// TIA Portal V18 export
FUNCTION "Pump Management" : Void   // FC44, LAD
{ S7_Optimized_Access := 'TRUE' }
VERSION : 0.1
// stored: AutoNumber false, IsIECCheckEnabled false, SetENOAutomatically false, UDAEnableTagReadback false
   VAR_TEMP
      mbit1 : Bool;
   END_VAR
BEGIN

REGION Network 1
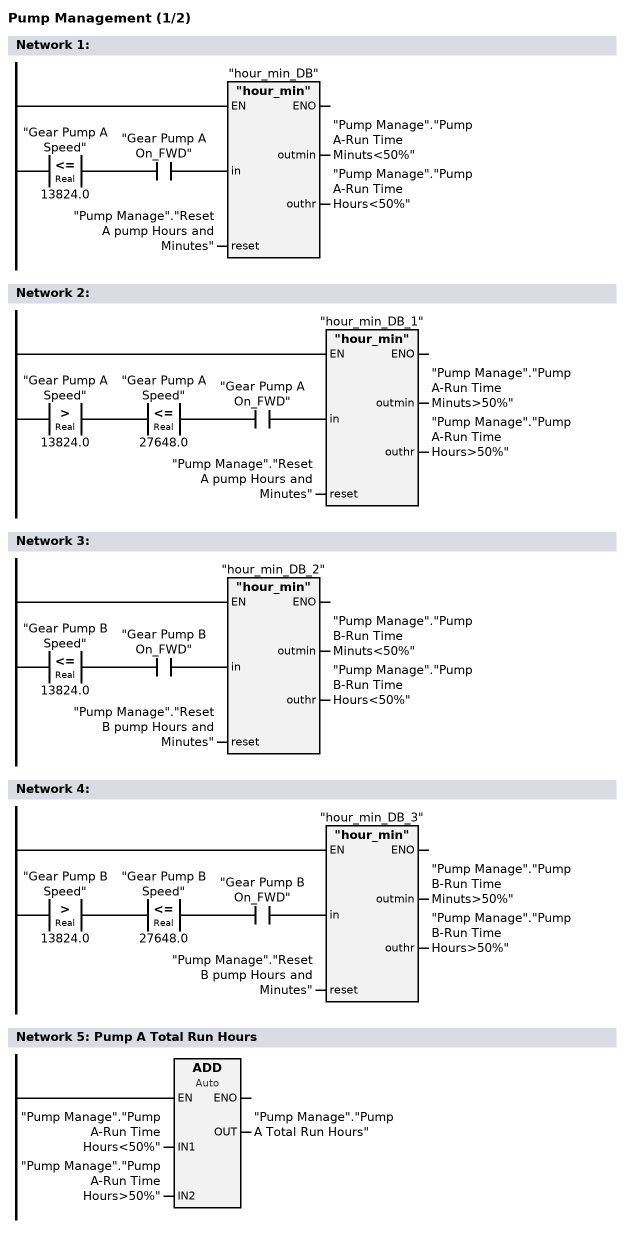
   RUNG wire#powerrail
      "hour_min_DB"(in := wire#w1, reset := "Pump Manage"."Reset A pump Hours and Minutes", outmin => "Pump Manage"."Pump A-Run Time Minuts<50%", outhr => "Pump Manage"."Pump A-Run Time Hours<50%")
   END_RUNG
   RUNG wire#powerrail
      { S7_Templates := "SrcType := Real" } LE_Contact(in1 := "Gear Pump A Speed", in2 := 13824.0)
      Contact( "Gear Pump A On_FWD" )
   END_RUNG wire#w1
   // the same network as SCL:
   "hour_min_DB"(in := ("Gear Pump A Speed" <= 13824.0) AND "Gear Pump A On_FWD",   // "hour_min"
                 reset := "Pump Manage"."Reset A pump Hours and Minutes",
                 outmin => "Pump Manage"."Pump A-Run Time Minuts<50%",
                 outhr => "Pump Manage"."Pump A-Run Time Hours<50%");
END_REGION

REGION Network 2
   RUNG wire#powerrail
      "hour_min_DB_1"(in := wire#w1, reset := "Pump Manage"."Reset A pump Hours and Minutes", outmin => "Pump Manage"."Pump A-Run Time Minuts>50%", outhr => "Pump Manage"."Pump A-Run Time Hours>50%")
   END_RUNG
   RUNG wire#powerrail
      { S7_Templates := "SrcType := Real" } GT_Contact(in1 := "Gear Pump A Speed", in2 := 13824.0)
      { S7_Templates := "SrcType := Real" } LE_Contact(in1 := "Gear Pump A Speed", in2 := 27648.0)
      Contact( "Gear Pump A On_FWD" )
   END_RUNG wire#w1
   // the same network as SCL:
   "hour_min_DB_1"(in := ("Gear Pump A Speed" > 13824.0) AND ("Gear Pump A Speed" <= 27648.0) AND "Gear Pump A On_FWD",   // "hour_min"
                   reset := "Pump Manage"."Reset A pump Hours and Minutes",
                   outmin => "Pump Manage"."Pump A-Run Time Minuts>50%",
                   outhr => "Pump Manage"."Pump A-Run Time Hours>50%");
END_REGION

REGION Network 3
   RUNG wire#powerrail
      "hour_min_DB_2"(in := wire#w1, reset := "Pump Manage"."Reset B pump Hours and Minutes", outmin => "Pump Manage"."Pump B-Run Time Minuts<50%", outhr => "Pump Manage"."Pump B-Run Time Hours<50%")
   END_RUNG
   RUNG wire#powerrail
      { S7_Templates := "SrcType := Real" } LE_Contact(in1 := "Gear Pump B Speed", in2 := 13824.0)
      Contact( "Gear Pump B On_FWD" )
   END_RUNG wire#w1
   // the same network as SCL:
   "hour_min_DB_2"(in := ("Gear Pump B Speed" <= 13824.0) AND "Gear Pump B On_FWD",   // "hour_min"
                   reset := "Pump Manage"."Reset B pump Hours and Minutes",
                   outmin => "Pump Manage"."Pump B-Run Time Minuts<50%",
                   outhr => "Pump Manage"."Pump B-Run Time Hours<50%");
END_REGION

REGION Network 4
   RUNG wire#powerrail
      "hour_min_DB_3"(in := wire#w1, reset := "Pump Manage"."Reset B pump Hours and Minutes", outmin => "Pump Manage"."Pump B-Run Time Minuts>50%", outhr => "Pump Manage"."Pump B-Run Time Hours>50%")
   END_RUNG
   RUNG wire#powerrail
      { S7_Templates := "SrcType := Real" } GT_Contact(in1 := "Gear Pump B Speed", in2 := 13824.0)
      { S7_Templates := "SrcType := Real" } LE_Contact(in1 := "Gear Pump B Speed", in2 := 27648.0)
      Contact( "Gear Pump B On_FWD" )
   END_RUNG wire#w1
   // the same network as SCL:
   "hour_min_DB_3"(in := ("Gear Pump B Speed" > 13824.0) AND ("Gear Pump B Speed" <= 27648.0) AND "Gear Pump B On_FWD",   // "hour_min"
                   reset := "Pump Manage"."Reset B pump Hours and Minutes",
                   outmin => "Pump Manage"."Pump B-Run Time Minuts>50%",
                   outhr => "Pump Manage"."Pump B-Run Time Hours>50%");
END_REGION

REGION Network 5: Pump A Total Run Hours
   RUNG wire#powerrail
      Add(in1 := "Pump Manage"."Pump A-Run Time Hours<50%", in2 := "Pump Manage"."Pump A-Run Time Hours>50%", out => "Pump Manage"."Pump A Total Run Hours")
   END_RUNG
   // the same network as SCL:
   "Pump Manage"."Pump A Total Run Hours" := "Pump Manage"."Pump A-Run Time Hours<50%" + "Pump Manage"."Pump A-Run Time Hours>50%";
END_REGION

REGION Network 6: Pump A Total Run Minutes
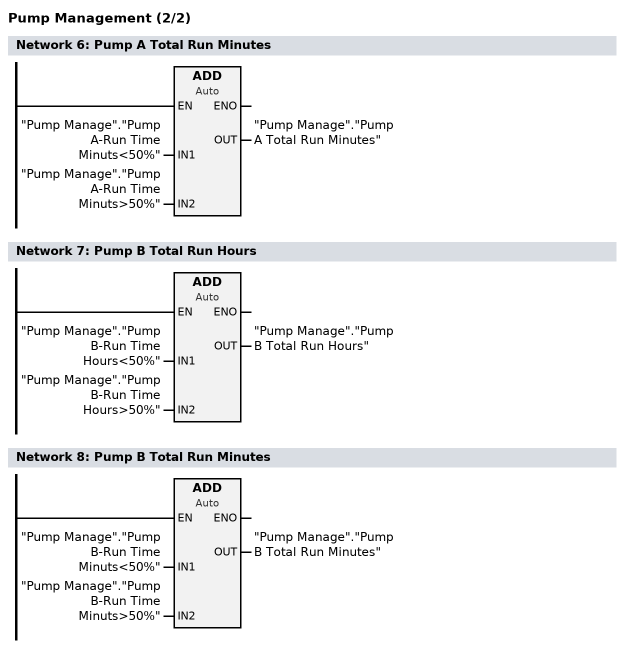
   RUNG wire#powerrail
      Add(in1 := "Pump Manage"."Pump A-Run Time Minuts<50%", in2 := "Pump Manage"."Pump A-Run Time Minuts>50%", out => "Pump Manage"."Pump A Total Run Minutes")
   END_RUNG
   // the same network as SCL:
   "Pump Manage"."Pump A Total Run Minutes" := "Pump Manage"."Pump A-Run Time Minuts<50%" + "Pump Manage"."Pump A-Run Time Minuts>50%";
END_REGION

REGION Network 7: Pump B Total Run Hours
   RUNG wire#powerrail
      Add(in1 := "Pump Manage"."Pump B-Run Time Hours<50%", in2 := "Pump Manage"."Pump B-Run Time Hours>50%", out => "Pump Manage"."Pump B Total Run Hours")
   END_RUNG
   // the same network as SCL:
   "Pump Manage"."Pump B Total Run Hours" := "Pump Manage"."Pump B-Run Time Hours<50%" + "Pump Manage"."Pump B-Run Time Hours>50%";
END_REGION

REGION Network 8: Pump B Total Run Minutes
   RUNG wire#powerrail
      Add(in1 := "Pump Manage"."Pump B-Run Time Minuts<50%", in2 := "Pump Manage"."Pump B-Run Time Minuts>50%", out => "Pump Manage"."Pump B Total Run Minutes")
   END_RUNG
   // the same network as SCL:
   "Pump Manage"."Pump B Total Run Minutes" := "Pump Manage"."Pump B-Run Time Minuts<50%" + "Pump Manage"."Pump B-Run Time Minuts>50%";
END_REGION
END_FUNCTION
